FUNCTION proj2_TupleStruct_2: LREAL
VAR_INPUT
    tuple: TupleStruct_2;
END_VAR


        proj2_TupleStruct_2 := tuple.field2;

END_FUNCTION

(* stored: ProductVersion 3.1.0.18, Version 1.1.0.1 *)
